{attribute 'linkalways'} 
{attribute 'no_explicit_call' := 'This FB is a CLASS and must be accessed using methods or properties'}
{attribute 'enable_dynamic_creation'}
FUNCTION_BLOCK Node_F_VN_MinElementElementwise_UINT EXTENDS VisionNode
VAR
    ipContainer : _ITcVnContainer;
    nMin : _UINT(0);
    hrPrev : _HRESULT(S_OK);
    hresult : _HRESULT(S_OK);
END_VAR

METHOD PUBLIC  Clone : I_Node
VAR
	pNode : POINTER TO Node_F_VN_MinElementElementwise_UINT;
END_VAR
pNode := __NEW(Node_F_VN_MinElementElementwise_UINT);
Clone := pNode^;
END_METHOD

METHOD FB_init : BOOL
VAR_INPUT
	bInitRetains : BOOL; // if TRUE, the retain variables are initialized (warm start / cold start)
	bInCopyCode : BOOL;  // if TRUE, the instance afterwards gets moved into the copy code (online change)
END_VAR
AddInput('ipContainer', ipContainer);
AddInput('nMin', nMin);
AddInput('hrPrev', hrPrev);
AddOutput('ipContainer', ipContainer);
AddOutput('hresult',hresult);
END_METHOD

METHOD PROTECTED OnExecute : HRESULT
hresult.Value := F_VN_MinElementElementwise_UINT(
    ipContainer := ipContainer.Value,
    nMin := nMin.Value,
    hrPrev:= hrPrev.Value);
END_METHOD

METHOD PUBLIC PreExecutionCheck
VAR_INPUT
	Check : I_PreExecutionChecks;
END_VAR
Check.IsTrue(ipContainer.IsValid, 'ipContainer must be a valid container');
END_METHOD

END_FUNCTION_BLOCK

(* stored: Version 1.1.0.1, ProductVersion 3.1.4024.13
   POU Node_F_VN_MinElementElementwise_UINT: Id {f455eaca-91ee-4288-ae04-423981b9442f}, SpecialFunc None
   Folder Constructor: Id {d5ea8cbb-8d93-4ad1-a2a8-1ed0735632f3}
   Method Clone: Id {4f76a7fa-cfd4-4568-ac99-a26483b26d37}
   Method FB_init: Id {0b785874-bcd3-40f3-827a-e07ea5317dc3}
   Method OnExecute: Id {68793877-bf54-4bea-aad7-c775ebf96b22}
   Method PreExecutionCheck: Id {ad760361-a133-4351-918c-d2deabd5890f} *)
